FUNCTION_BLOCK E_STOP
  (* Version 1.0, 2005-12-19, Goran Cengic, Chalmers *)
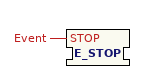
  EVENT_INPUT
    STOP;
  END_EVENT
  EC_STATES
    S0;
  END_STATES
END_FUNCTION_BLOCK
